(* This testsuite tests the function block FB_AdjustAssertFailureMessageToMax255CharLength_Test *)
{attribute 'call_after_init'}
FUNCTION_BLOCK FB_AdjustAssertFailureMessageToMax252CharLength_Test EXTENDS TcUnit.FB_TestSuite

TestInstancePath252CharsExpectTooLongTestInstancePath();
TestInstancePath220CharsExpectShortenedTestInstancePath();
TestInstancePath255CharsExpectTooLongTestInstancePath();

METHOD TestInstancePath220CharsExpectShortenedTestInstancePath
VAR
    AdjustAssertFailureMessageToMax252CharLength : FB_AdjustAssertFailureMessageToMax252CharLength;

    // @Text-Fixture
    TestInstancePathNameWith220Chars : Tc2_System.T_MaxString := 'PRG_TEST.LongInstanceNameLongInstanceNameLongInstanceNameLongInstanceNameLongInstanceNameLongInstanceNameLongInstanceNameLongInstanceNameLongInstanceNameLongInstanceName@LONGTESTNAMELONGTESTNAMELONGTESTNAMELONGTESTNAMELO';
    TooLongTestMessage60Chars : Tc2_System.T_MaxString := 'Very long message that is 60 characters long which means tha';
    
    // @Test-Result-Expected
    // 220 + 32 = 252 (in other words, expected test message should be 32 characters long including '...TestMsg too long'
    TestMessageResultExpected : Tc2_System.T_MaxString := 'Very long mes...TestMsg too long'; 

    // @Test-Result
    TestInstancePathResult : Tc2_System.T_MaxString;
    TestMessageResult : Tc2_System.T_MaxString;
END_VAR
TEST('TestInstancePath220CharsExpectShortenedTestInstancePath');


AdjustAssertFailureMessageToMax252CharLength(MsgFmtString := TestInstancePathNameWith220Chars,
                                             StringArg := TooLongTestMessage60Chars,
                                             MsgFmtStringProcessed => TestInstancePathResult,
                                             StringArgProcessed => TestMessageResult);


AssertEquals_STRING(Expected := TestInstancePathNameWith220Chars, // Same test instance path should be expected as the one going in
                    Actual := TestInstancePathResult,
                    'Test instance path not correct');

AssertEquals_STRING(Expected := TestMessageResultExpected,
                    Actual := TestMessageResult,
                    'Test message not correct');

TEST_FINISHED();
END_METHOD

METHOD PRIVATE TestInstancePath252CharsExpectTooLongTestInstancePath
VAR
    AdjustAssertFailureMessageToMax252CharLength : FB_AdjustAssertFailureMessageToMax252CharLength;

    // @Text-Fixture
    TestInstancePathNameWith252Chars : Tc2_System.T_MaxString := 'PRG_TEST.LongInstanceNameLongInstanceNameLongInstanceNameLongInstanceNameLongInstanceNameLongInstanceNameLongInstanceNameLongInstanceNameLongInstanceNameLongInstanceName@LONGTESTNAMELONGTESTNAMELONGTESTNAMELONGTESTNAMELONGTESTNAMELONGTESTNAMELONGTESTNA';
    ShortTestMessage : Tc2_System.T_MaxString := 'Very short message';

    // @Test-Result-Expected
    TestInstancePathNameWith252CharsExpectedResult : Tc2_System.T_MaxString := 'PRG_TEST.LongInstanceNameLongInstanceNameLongInstanceNameLongInstanceNameLongInstanceNameLongInstanceNameLongInstanceNameLongInstanceNameLongInstanceNameLongInstanceName@LONGTESTNAMELONGTESTNAMELONGTESTNAMELONGTESTNAMELONGTESTNAMELO...TestName too long';
    ShortTestMessageExpectedResult : Tc2_System.T_MaxString := '';
    
    // @Test-Result
    TestInstancePathNameWith252CharsResult : Tc2_System.T_MaxString;
    ShortTestMessageResult : Tc2_System.T_MaxString;
END_VAR
TEST('TestInstancePath252CharsExpectTooLongTestInstancePath');

AdjustAssertFailureMessageToMax252CharLength(MsgFmtString := TestInstancePathNameWith252Chars,
                                             StringArg := ShortTestMessage,
                                             MsgFmtStringProcessed => TestInstancePathNameWith252CharsResult,
                                             StringArgProcessed => ShortTestMessageResult);

AssertEquals_STRING(Expected := TestInstancePathNameWith252CharsExpectedResult,
                    Actual := TestInstancePathNameWith252CharsResult,
                    'Test instance path not correct');

AssertEquals_STRING(Expected := ShortTestMessageExpectedResult,
                    Actual := ShortTestMessageResult,
                    'Test message not correct');

TEST_FINISHED();
END_METHOD

METHOD PRIVATE TestInstancePath255CharsExpectTooLongTestInstancePath
VAR
    AdjustAssertFailureMessageToMax252CharLength : FB_AdjustAssertFailureMessageToMax252CharLength;

    // @Text-Fixture
    TestInstancePathNameWith255Chars : Tc2_System.T_MaxString := 'PRG_TEST.LongInstanceNameLongInstanceNameLongInstanceNameLongInstanceNameLongInstanceNameLongInstanceNameLongInstanceNameLongInstanceNameLongInstanceNameLongInstanceName@LONGTESTNAMELONGTESTNAMELONGTESTNAMELONGTESTNAMELONGTESTNAMELONGTESTNAMELONGTESTNAGAV';
    ShortTestMessage : Tc2_System.T_MaxString := 'Very short message';

    // @Test-Result-Expected
    TestInstancePathNameWith252CharsExpectedResult : Tc2_System.T_MaxString := 'PRG_TEST.LongInstanceNameLongInstanceNameLongInstanceNameLongInstanceNameLongInstanceNameLongInstanceNameLongInstanceNameLongInstanceNameLongInstanceNameLongInstanceName@LONGTESTNAMELONGTESTNAMELONGTESTNAMELONGTESTNAMELONGTESTNAMELO...TestName too long';
    ShortTestMessageExpectedResult : Tc2_System.T_MaxString := '';

    // @Test-Result
    TestInstancePathNameWith252CharsResult : Tc2_System.T_MaxString;
    ShortTestMessageResult : Tc2_System.T_MaxString;
END_VAR
TEST('TestInstancePath255CharsExpectTooLongTestInstancePath');

AdjustAssertFailureMessageToMax252CharLength(MsgFmtString := TestInstancePathNameWith255Chars,
                                             StringArg := ShortTestMessage,
                                             MsgFmtStringProcessed => TestInstancePathNameWith252CharsResult,
                                             StringArgProcessed => ShortTestMessageResult);

AssertEquals_STRING(Expected := TestInstancePathNameWith252CharsExpectedResult,
                    Actual := TestInstancePathNameWith252CharsResult,
                    'Test instance path not correct');

AssertEquals_STRING(Expected := ShortTestMessageExpectedResult,
                    Actual := ShortTestMessageResult,
                    'Test message not correct');

TEST_FINISHED();
END_METHOD

END_FUNCTION_BLOCK

(* stored: Version 1.1.0.1, ProductVersion 3.1.4022.18
   POU FB_AdjustAssertFailureMessageToMax252CharLength_Test: Id {305341a5-f462-4bcb-ba17-ae2773c50e69}, SpecialFunc None
   Method TestInstancePath220CharsExpectShortenedTestInstancePath: Id {dc008964-f701-440f-97f6-bba60a51fe93}
   Method TestInstancePath252CharsExpectTooLongTestInstancePath: Id {f67e3ff5-02f7-4268-9fa7-f06935f8269a}
   Method TestInstancePath255CharsExpectTooLongTestInstancePath: Id {fbb2640b-9b30-45ae-a207-49da858d57e9} *)
